# B&R Automation Studio project Vis
Automation Studio 4.9.3.144 SP

## Configuration Config1

CPU X20CP1382, AutomationRuntime B4.83, Build 4.1.2, Vc V4.72.2

### Hardware
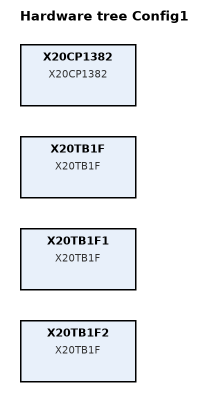
```
X20CP1382 : X20CP1382 v1.11.0.0  [X1 -> X1.SL; X2 -> X2.SL; X3 -> X3.SL]
  Module X1 (Type=X1, Virtual=true, Version=1.11.0.0)
    Connection (Connector=SS1, TargetModule=X20TB1F, TargetConnector=SS)
    Connection (Connector=SL, TargetModule=X20CP1382, TargetConnector=X1)
  Module X2 (Type=X2, Virtual=true, Version=1.11.0.0)
    Connection (Connector=SS1, TargetModule=X20TB1F1, TargetConnector=SS)
    Connection (Connector=SL, TargetModule=X20CP1382, TargetConnector=X2)
  Module X3 (Type=X3, Virtual=true, Version=1.11.0.0)
    Connection (Connector=SS1, TargetModule=X20TB1F2, TargetConnector=SS)
    Connection (Connector=SL, TargetModule=X20CP1382, TargetConnector=X3)
  Connector IF2:
    ActivateDevice = 1
    Vnc1
    VncVcObjectName1 = Visu
    VncKeyMappingFile1 = VC\PS2-Keyboard.dis
    VncAuthentication1 = 1
    VncPasswordViewOnly1 = v
    VncPasswordViewControl1 = c
    VncMaxConnections1 = 10
    VncRefreshRate1 = 300
  ConfigurationID = Vis_Config1
  Simulation = 1
X20TB1F : X20TB1F v1.0.0.0
X20TB1F1 : X20TB1F v1.0.0.0
X20TB1F2 : X20TB1F v1.0.0.0
```

## Logical view

- Visualisation Logical/Visu (not shown)

### Program Logical/Program (IEC)

#### Types.typ
```iecst
TYPE
	krok :
		(
		zielone,
		OFF,
		noc_zolte,
		NOC,
		czekaj,
		zolto_czerwone,
		czerwone,
		zolte
		);
END_TYPE
```

#### Variables.var
```iecst
VAR
	zolte1 : BOOL;
	czerwone1 : BOOL;
	zielone1 : BOOL;
	zolte2 : BOOL;
	czerwone2 : BOOL;
	zielone2 : BOOL;
	stan : krok;
	TON_Zielone : TON;
	TON_Zolte : TON;
	TON_Czerwone : TON;
	swiatlo : krok;
	przycisk : BOOL;
	noc : BOOL;
	noc0 : BOOL;
	start : BOOL;
	czekaj_ : BOOL;
	kolory_nocy : INT;
	TON_AUTA : TON;
	auta1 : INT;
	auta2 : INT;
	licznik : INT;
END_VAR
```

#### Main.st
```iecst
PROGRAM _INIT
	(* Insert code here *)

END_PROGRAM

PROGRAM _CYCLIC
	(* Insert code here *)
	//jeżeli nastała noc
	IF noc AND NOT noc0 THEN
		stan := NOC;
	END_IF;

	//Jeżeli kliknęliśmy start i dopiero uruchamiamy sygnalizację
	IF stan = OFF AND start THEN
		stan := zolte;//zapal żółte
	//Jeżeli nie jest kliknięty Start wyłączamy sygnalizację
	ELSIF NOT start THEN
		stan := OFF;
	END_IF;

	//ustawienie timera dodającego auta na 400 ms
	TON_AUTA.PT := T#400ms;
	TON_AUTA.IN := 1;

	//Jeżeli minęło 400 ms
	IF TON_AUTA.Q THEN
		//Jeżeli jest noc
		IF noc THEN
			IF auta1>0 AND (licznik = 2 OR licznik = 4 OR licznik = 6) THEN
				auta1 := auta1 -1;
			END_IF;
			IF auta2>0 AND (licznik = 1 OR licznik = 3 OR licznik = 5) THEN
				auta2 := auta2 -1;
			END_IF;
			IF licznik = 2  THEN
				auta1 := auta1 + 2;
			END_IF;
			IF licznik = 6  THEN
				auta2 := auta2 + 2;
				licznik := 0;
			END_IF;
		//Jeżeli jest dzień
		ELSE
			IF licznik >= 3  THEN
				auta1 := auta1 + 2;
				auta2 := auta2 + 1;
				licznik := 0;
			END_IF;
			CASE stan OF
				zielone:
					IF auta1>1 THEN
						auta1 := auta1 -2;
					END_IF;
				czerwone:
					IF auta2>1 THEN
						auta2 := auta2 -2;
					END_IF;
				czekaj:
					IF swiatlo = 2 AND auta1>1 THEN
						auta1 := auta1 -2;
					ELSIF swiatlo = 4 AND auta2 >1 THEN
						auta2 := auta2 -2;
					END_IF;
			END_CASE;
		END_IF;
		licznik := licznik + 1;
		TON_AUTA.IN := 0;
	END_IF;

	//maszyna stanów
	CASE stan OF
		OFF:
			zielone1 := 0;
			zolte1 := 0;
			czerwone1 := 0;
			zielone2 := 0;
			zolte2 := 0;
			czerwone2 := 0;

			TON_Zielone.IN := 0;
			TON_Zolte.IN := 0;
			TON_Czerwone.IN := 0;
		zielone:
			zielone1:= 1;
			zolte1 := 0;
			czerwone1:= 0;

			zielone2 := 0;
			zolte2 := 0;
			czerwone2 := 1;

			TON_Zielone.PT := T#5s;
			TON_Zielone.IN := 1;
			IF TON_Zielone.Q THEN
				stan := czekaj;
				swiatlo := zolte;//zapamiętanie następnego kroku
				TON_Zielone.IN := 0;
			END_IF;
		zolte:
			zielone1 :=0;
			zolte1 := 1;
			czerwone1 := 0;

			zielone2 := 0;
			zolte2 := 1;
			czerwone2 := 1;

			TON_Zolte.PT := T#1s;
			TON_Zolte.IN := 1;
			IF TON_Zolte.Q THEN
				stan := czerwone;
				TON_Zolte.IN := 0;
			END_IF;

		czerwone:
			zielone1 := 0;
			zolte1 := 0;
			czerwone1 := 1;

			zielone2 := 1;
			zolte2 := 0;
			czerwone2 := 0;

			TON_Czerwone.PT := T#5s;
			TON_Czerwone.IN := 1;
			IF TON_Czerwone.Q THEN
				stan := czekaj;
				swiatlo := zolto_czerwone;//zapamiętanie następnego kroku
				TON_Czerwone.IN := 0;
			END_IF;

		zolto_czerwone:
			zielone1 :=0;
			zolte1 := 1;
			czerwone1 := 1;

			zielone2 := 0;
			zolte2 := 1;
			czerwone2 := 0;

			TON_Zolte.PT := T#1s;
			TON_Zolte.IN := 1;
			IF TON_Zolte.Q THEN
				stan := zielone;
				TON_Zolte.IN := 0;
			END_IF;
		czekaj:
			czekaj_ := TRUE;
			IF przycisk THEN
				stan := swiatlo;
				przycisk := FALSE;
				czekaj_ := FALSE;
			END_IF;
		NOC:
			zielone1 := 0;
			zolte1 := 0;
			czerwone1 := 0;
			zielone2 := 0;
			zolte2 := 0;
			czerwone2 := 0;

			TON_Zolte.PT := T#1s;
			TON_Zolte.IN := 1;
			IF TON_Zolte.Q THEN
				stan := noc_zolte;
				TON_Zolte.IN := 0;
			END_IF;
		noc_zolte:
			zielone1 := 0;
			zolte1 := 1;
			czerwone1 := 0;
			zielone2 := 0;
			zolte2 := 1;
			czerwone2 := 0;

			TON_Zolte.PT := T#1s;
			TON_Zolte.IN := 1;
			IF TON_Zolte.Q THEN
				stan := NOC;
				TON_Zolte.IN := 0;
			END_IF;
			IF NOT noc THEN
	  			stan := zolte;
			END_IF;

	END_CASE;
	//przypisanie obecnego stanu zmiennej noc do zmiennej noc0
	noc0 := noc;
	IF noc THEN
		kolory_nocy := 213;
	ELSE
		kolory_nocy := 187;
	END_IF;

	//uruchomienie timerów
	TON_Zielone ();
	TON_Zolte();
	TON_Czerwone();
	TON_AUTA();
END_PROGRAM

PROGRAM _EXIT
	(* Insert code here *)

END_PROGRAM
```

Listed in the project but not available here: Logical/Global.typ, Logical/Global.var, Logical/Libraries
